{attribute addProperty BoxType "KL1202"}
{attribute addProperty Id "Channel_1Channel_DCE4399300Channel_2Channel_DCE4399300"}
{attribute addProperty CRC "323723758"}
{attribute addProperty SizeInBites "0"}
{attribute addProperty SizeInBytes "0"}
TYPE KL1202_134BA1EE :
STRUCT
	{attribute addProperty Name "Channel_1"}
	Channel_1 : Channel_DCE43993;
	{attribute addProperty Name "Channel_2"}
	Channel_2 : Channel_DCE43993;
END_STRUCT
END_TYPE

(* stored: Version 1.2.0.0, ProductVersion 3.1.4024.9
   DUT KL1202_134BA1EE: Id {e006086e-9326-47e7-a0d4-0e6ae5c61e1a} *)
